(* CoDeSys 2.3.9.62 project: 0750-0849.WagoAppKNX.SunshadeActuator.pro *)
(* Libraries: C:\Work\WAGO\WAGO.Sandbox\WAGO.KNX\CoDeSys\2.3\mod_com.lib, C:\Work\WAGO\WAGO.Sandbox\WAGO.KNX\CoDeSys\2.3\KNX_Standard.lib*27.4.23 16:22:16, WAGOLibKNXDevice.lib 23.1.08 13:40:44, C:\Work\WAGO\WAGO.Sandbox\WAGO.KNX\CoDeSys\2.3\KNX_IP_750_849_01.lib*2.5.23 10:23:28, SysLibGetAddress.lib 7.9.10 15:37:47, C:\Work\WAGO\WAGO.Sandbox\WAGO.KNX\CoDeSys\2.3\KNX_Applikations_02.lib*27.4.23 16:22:16, C:\Work\WAGO\WAGO.Sandbox\WAGO.KNX\CoDeSys\2.3\DALI_02.lib*27.4.23 16:22:16, Standard.lib, SYSLIBCALLBACK.LIB, WagoLibSockets.lib 11.4.05 09:27:06, SysLibSockets.lib 16.10.01 08:59:11, NETVARUDP_LIB_V23.LIB 8.11.10 12:37:48 *)

(* PLC configuration (modules and I/O channels)
AT %IB0 [BYTEOnB_I] First Byte of 24
AT %QB0 [BYTEOnB_Q] First Byte of 24
Fieldbus variables [FB_VARS] node 1, in %IB0 out %QB0
Flag variables [FLAG_VARS] node 2, in %IB0 out %QB0
Modbus-Master [MB_MASTER] node 3, in %IB0 out %QB0
*)

(* Global variable list: Networkmanagement implicit Variables UDP *)
VAR_GLOBAL CONSTANT
	USE_NWVARS_UDP : BOOL := FALSE;
	MAX_NetVarItems_UDP	: INT := 0;
	MAX_NetVarPDO_Rx_UDP	: INT := 0;
	MAX_NetVarPDO_Tx_UDP	: INT := 0;
	MAX_NetVarOD_UDP		: INT := 0;
END_VAR
VAR_GLOBAL
	pNetVarItems_UDP		: ARRAY[0..MAX_NetVarItems_UDP] OF NetVarDataItem_UDP;
	pNetVarPDO_Rx_UDP		: ARRAY[0..MAX_NetVarPDO_Rx_UDP] OF NetVarPDO_Rx_UDP;
	pNetVarPDO_Tx_UDP		: ARRAY[0..MAX_NetVarPDO_Tx_UDP] OF NetVarPDO_Tx_UDP;
	pNetVarOD_UDP			: ARRAY[0..MAX_NetVarOD_UDP] OF NetVarSDO_UDP;
	pNetVarPDO_Rx_Diagnosis_UDP : ARRAY[0..MAX_NetVarPDO_Rx_UDP] OF NetVarUDPDiagStruct;
	pNetVarPDO_Tx_Diagnosis_UDP : ARRAY[0..MAX_NetVarPDO_Tx_UDP] OF NetVarUDPDiagStruct;
END_VAR

(* POU PLC_PRG, CFC *)
PROGRAM PLC_PRG
VAR
END_VAR
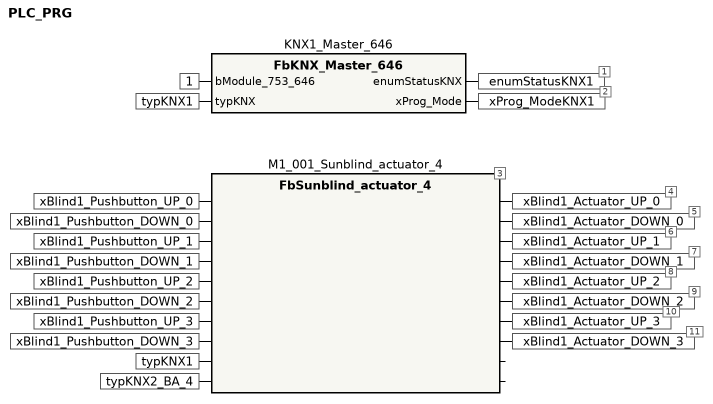
_CFC_ (* Continuous Function Chart, elements in execution order *)
#0 KNX1_Master_646:FbKNX_Master_646(bModule_753_646: 1, typKNX: typKNX1)
#1 enumStatusKNX1 <= #0.enumStatusKNX
#2 xProg_ModeKNX1 <= #0.xProg_Mode
#3 M1_001_Sunblind_actuator_4:FbSunblind_actuator_4(xBlind1_Pushbutton_UP_0, xBlind1_Pushbutton_DOWN_0, xBlind1_Pushbutton_UP_1, xBlind1_Pushbutton_DOWN_1, xBlind1_Pushbutton_UP_2, xBlind1_Pushbutton_DOWN_2, xBlind1_Pushbutton_UP_3, xBlind1_Pushbutton_DOWN_3, typKNX1, typKNX2_BA_4)
#4 xBlind1_Actuator_UP_0 <= #3.out 1
#5 xBlind1_Actuator_DOWN_0 <= #3.out 2
#6 xBlind1_Actuator_UP_1 <= #3.out 3
#7 xBlind1_Actuator_DOWN_1 <= #3.out 4
#8 xBlind1_Actuator_UP_2 <= #3.out 5
#9 xBlind1_Actuator_DOWN_2 <= #3.out 6
#10 xBlind1_Actuator_UP_3 <= #3.out 7
#11 xBlind1_Actuator_DOWN_3 <= #3.out 8
_END_CFC_
END_PROGRAM

(* Visualisation Visualisierung
embedded screen at (0,0)-(801,601): Sunblind_actuator_visu
*)
